// TIA Portal V17 export
// export: Created 2021-12-03T08:13:03.6409176Z, ExportSetting WithDefaults, DisplayName Totally Integrated Automation Portal, DisplayVersion V17, DisplayName TIA Portal Openness, DisplayVersion V17, DisplayName TIA Portal Version Control Interface, DisplayVersion V17, DisplayName STEP 7 Professional, DisplayVersion V17, DisplayName STEP 7 Safety, DisplayVersion V17, DisplayName WinCC Advanced, DisplayVersion V17
DATA_BLOCK "GDB_Acc_Ctrl"   // DB63
VERSION : 0.1
// stored: AutoNumber false, IsOnlyStoredInLoadMemory false, IsWriteProtectedInAS false
   VAR
      Acc : Struct
         RdyDly : Bool;   // Готовность ускорителя
         RdyOff : Bool;
         RdyTm : Bool;
         CondIntrlc : Bool;   // Условия для интерлока
         Chil_PwrOn : Bool;   // Контактор. Питание модуля охлаждения
         AccCsPrehOn : Bool;   // Пускатель. Питание сушки ускорителя
         DetLine_ChilPwrOn : Bool;   // Контактор. Питание климатической системы. Детекторная линейка 1
         DetLine_RelayOn : Bool;   // Контактор. Питание системы управления детекторной линейки
         Mod380V_RlyOn : Bool;   // Включение питания 380В модулятора.
         AccMod220V_PwrOn : Bool;   // Включение питания ускорителя и модулятора 220В
         Acc220V_PwrOn : Bool;   // Включение питания ускорителя 220В
         ChilOnDly : Bool;   // Задержка включения чиллера
         ChilOffDly : Bool;   // Задержка выключения чиллера
         RFXrayChilTmOk : Bool;   // Задержка на охлаждение между сканированиями
         AccSigFault : Bool;   // Ошибка ускорителя
         RFXrayChilTm : Time;   // Прошедешее время охлаждения ускорителя
         ActState : Int;
         "X-RayOn" : Bool;
         State : Struct
            Bit08_AccE_Stop { ExternalVisible := 'False'; ExternalWritable := 'False'} : Bool;   // 1=E-stop accelerator control console / Accelerator Control Statusword 1 / Аварийная кнопка на ускорителе
            Bit09_Stdby { ExternalVisible := 'False'; ExternalWritable := 'False'} : Bool;   // 1=Stand by / 1=Warning / Пауза
            Bit10_RFOn { ExternalVisible := 'False'; ExternalWritable := 'False'} : Bool;   // 1=RF On / Spare / СВЧ излучение
            Bit11_HiDoseOn { ExternalVisible := 'False'; ExternalWritable := 'False'} : Bool;   // 1=High dose On / Spare / ТИ включено
            Bit12_Accelerator_GrpCirBr_Flt { ExternalVisible := 'False'; ExternalWritable := 'False'} : Bool;   // Spare / 1=Ready For Scanning / 1 = Ошибка по питанию группы ускоритель
            Bit13_AccSig_RemKey { ExternalVisible := 'False'; ExternalWritable := 'False'} : Bool;   // Spare / State: 1=Error
            Bit14 { ExternalVisible := 'False'; ExternalWritable := 'False'} : Bool;   // Spare / State: 1=Service mode
            Bit15 { ExternalVisible := 'False'; ExternalWritable := 'False'} : Bool;   // Spare / 1=Fault
            Bit00_RemMdSel { ExternalVisible := 'False'; ExternalWritable := 'False'} : Bool;   // 1=Remote mode selected / 1=E-stop accelerator
            Bit01_PwrOnSts { ExternalVisible := 'False'; ExternalWritable := 'False'} : Bool;   // 1=Power On / 1=No Group Fault Chiller / Питание ВКЛ
            Bit02_WarmUp { ExternalVisible := 'False'; ExternalWritable := 'False'} : Bool;   // 1=Warming Up / Remote Interlock 1 / Прогрев
            Bit03_Clear { ExternalVisible := 'False'; ExternalWritable := 'False'} : Bool;   // 1=Clear / Spare / Предварительная готовность
            Bit04_Rdy { ExternalVisible := 'False'; ExternalWritable := 'False'} : Bool;   // 1=Ready / Spare / Основная готовность
            Bit05_XrayOn { ExternalVisible := 'False'; ExternalWritable := 'False'} : Bool;   // 1=X-Ray On / Detector Line: Trigger rate / Тормозное излучение
            Bit06_Flt { ExternalVisible := 'False'; ExternalWritable := 'False'} : Bool;   // 1=Fault / Spare / Ошибка
            Bit07_AccPanelE_Stop { ExternalVisible := 'False'; ExternalWritable := 'False'} : Bool;   // 1=E-stop accelerator / Spare / Аварийная кнопка на консоли
         END_STRUCT;
      END_STRUCT;
      Chill : Struct
         OffTmLowSel : Bool;   // Выбрано короткое время выключения
         OnTmLowSel : Bool;   // Выбрано короткое время включения
      END_STRUCT;
      AxTRIG : Struct
         AccOn : Bool;
         AccOff : Bool;
         SAreaCls : Bool;
      END_STRUCT;
      AxSR : Struct
         AccRdy : Bool;
      END_STRUCT;
      IntrlckAcc : Bool;
   END_VAR
BEGIN
END_DATA_BLOCK
